TYPE ST_Timer :
STRUCT
	StartTimer : BOOL := TRUE;
	TimeToPass : TIME;
	CurrentTime : TIME;
	IsFinished : BOOL := FALSE;
END_STRUCT
END_TYPE

(* stored: Version 1.1.0.1, ProductVersion 3.1.4024.12
   DUT ST_Timer: Id {a910b9e0-07ef-4358-bc86-e06d82264ede} *)
